FUNCTION_BLOCK EtherCATFactory
VAR

END_VAR

METHOD PUBLIC CreateEtherCATDevice : I_EtherCATDevice
VAR_INPUT
END_VAR

VAR
	devicePtr: POINTER TO EtherCATDevice;
END_VAR
devicePtr := __NEW(EtherCATDevice);
CreateEtherCATDevice := devicePtr^;
END_METHOD

END_FUNCTION_BLOCK

(* stored: Version 1.1.0.1, ProductVersion 3.1.4024.12
   POU EtherCATFactory: Id {068d6bf7-c72d-464f-947f-295d84e58383}, SpecialFunc None
   Method CreateEtherCATDevice: Id {76de9ec2-3bf9-4c3c-bb39-afd82b7c6d29} *)
